//{attribute 'qualified_only'}
VAR_GLOBAL
	A1_Arm1Mode:ARRAY[1..2,0..8] OF BOOL; //-----modify1118
	A1_Arm1Mode_Mid:ARRAY[1..2,0..8] OF BOOL;
    A1_Arm1Mode_TRIG:ARRAY[1..2,0..8] OF  R_TRIG;
	A1_Arm1ModeL:ARRAY[1..2,0..8] OF BOOL;
    A1_Arm1Mode_F_TRIG:ARRAY[1..4,0..6] OF  F_TRIG;
END_VAR

(* stored: Version 1.1.0.1, ProductVersion 3.1.4024.11
   GVL GVL_HmiMid: Id {64e88e01-f0c9-4682-9994-b5aa2920e88c} *)
